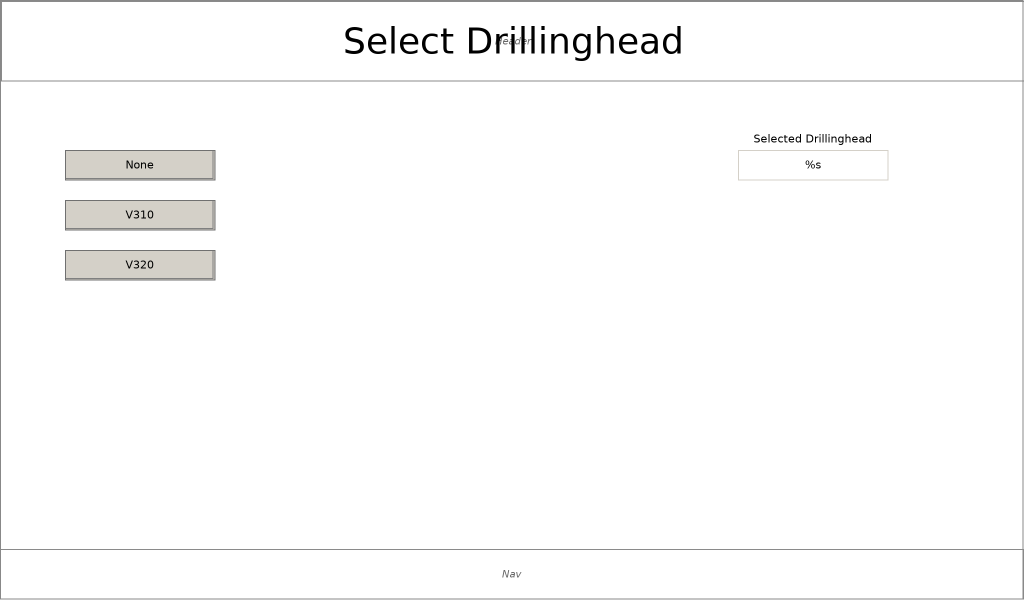
VISUALIZATION SelectDrillinghead  // 1024x600
    Frame (1,1 1024x80)
        shows Header()
    Frame (0,549 1024x50)
        shows Nav()
    Label (335,17 357x48), "Select Drillinghead"
    Textfield (738,150 150x30), "%s", text variable: Motion.sSelectedDrillingheadType
    Label (738,124 150x30), "Selected Drillinghead"
    Button (65,150 150x30), "None"
        OnMouseDown: execute { Motion.bNone := TRUE; }
        OnMouseUp: execute { Motion.bNone := FALSE; }
    Button (65,200 150x30), "V310"
        OnMouseDown: execute { Motion.bV310 := TRUE; }
        OnMouseUp: execute { Motion.bV310 := FALSE; }
    Button (65,250 150x30), "V320"
        OnMouseDown: execute { Motion.bV320 := TRUE; }
        OnMouseUp: execute { Motion.bV320 := FALSE; }
END_VISUALIZATION

(* stored: Version 1.1.0.1, ProductVersion 3.1.4024.12
   Visu SelectDrillinghead: Id {5c4773c5-8272-4e74-86b5-1c82087e8252} *)
